Fanuc KAREL source: wpathresenb.kl

PROGRAM wpathresenb
%NOLOCKGROUP
VAR
  p : POSITION
  q : POSITION
  i : INTEGER
  r : REAL
BEGIN
  WITH $PATHRES_ENB = TRUE MOVE TO p
END wpathresenb
